// TIA Portal V20 export
DATA_BLOCK "PM03"   // DB219
// stored: MemoryReserve 100
   VAR
      "C12 UNWINDER SPLICER HOLDER SPLICING LEFT MODULE MOVER FORWARD" : Bool;
      "C12 UNWINDER SPLICER HOLDER SPLICING LEFT MODULE MOVER BACKWARD" : Bool;
      "C13 UNWINDER SPLICER HOLDER SPLICING RIGHT MODULE MOVER FORWARD" : Bool;
      "C13 UNWINDER SPLICER HOLDER SPLICING RIGHT MODULE MOVER BACKWARD" : Bool;
      "C14 UNWINDER SPLICER HOLDER ELECTRODE LEFT HOLDER MODULE MOVER FORWARD" : Bool;
      "C14 UNWINDER SPLICER HOLDER ELECTRODE LEFT HOLDER MODULE MOVER BACKWARD" : Bool;
      "C15 UNWINDER SPLICER HOLDER ELECTRODE RIGHT HOLDER MODULE MOVER FORWARD" : Bool;
      "C15 UNWINDER SPLICER HOLDER ELECTRODE RIGHT HOLDER MODULE MOVER BACKWARD" : Bool;
      "C16 UNWINDER SPLICER TAPE LOADING TURN ROTATE" : Bool;
      "C16 UNWINDER SPLICER TAPE LOADING TURN HOME" : Bool;
      "C17 UNWINDER SPLICER TAPE ATTACH UNIT FORWARD" : Bool;
      "C17 UNWINDER SPLICER TAPE ATTACH UNIT BACKWARD" : Bool;
      SPARE_1 : Bool;
      SPARE_2 : Bool;
      SPARE_3 : Bool;
      SPARE_4 : Bool;
   END_VAR
BEGIN
END_DATA_BLOCK
